// TIA Portal V20 export
FUNCTION_BLOCK "GM_ReceiveFData"   // FB116, LAD
TITLE = Template: GM sending data
// Template v0.1
// stored: MemoryReserve 100, Namespace Safety, SetENOAutomatically false
   VAR_INPUT
      Connection_ID_Send : Word;
      Connection_ID_Receive : Word;
      Send_Ack_Rcv_Length : UInt;
      Receive_Rcv_Length : UInt;
   END_VAR
   VAR_IN_OUT
      RcvBuffer : Array[0..1, 0..121] of Byte;   // Temporary receive buffer: Max Rcv-Array of F-Link Communication Length = 122 Bytes
      ReceivedData : Array[0..121] of Byte;   // Received raw data from PLC 2
      ReceivedAck : Array[0..121] of Byte;   // Received acknowledge data for communication PLC 1 to PLC 2
   END_VAR
   VAR
      instTRcvAck { S7_SetPoint := 'True'} : TRCV;   // Receive acknowledge data from PLC2
      instTRcvData { S7_SetPoint := 'True'} : TRCV;   // Receive data from PLC2
      statErrorRcvAck { S7_SetPoint := 'True'} : Word;   // variable for saving the status of TRCV block in case of error
      statErrorRcvData : Word;   // variable for saving the status of TRCV block in case of error
   END_VAR
BEGIN

REGION Network 1: Receive ACK_RCV_ARRAY from Plc1ToPlc2 Communication / Receive Acknowledge signal from partner
   // receive ack. signal from each station
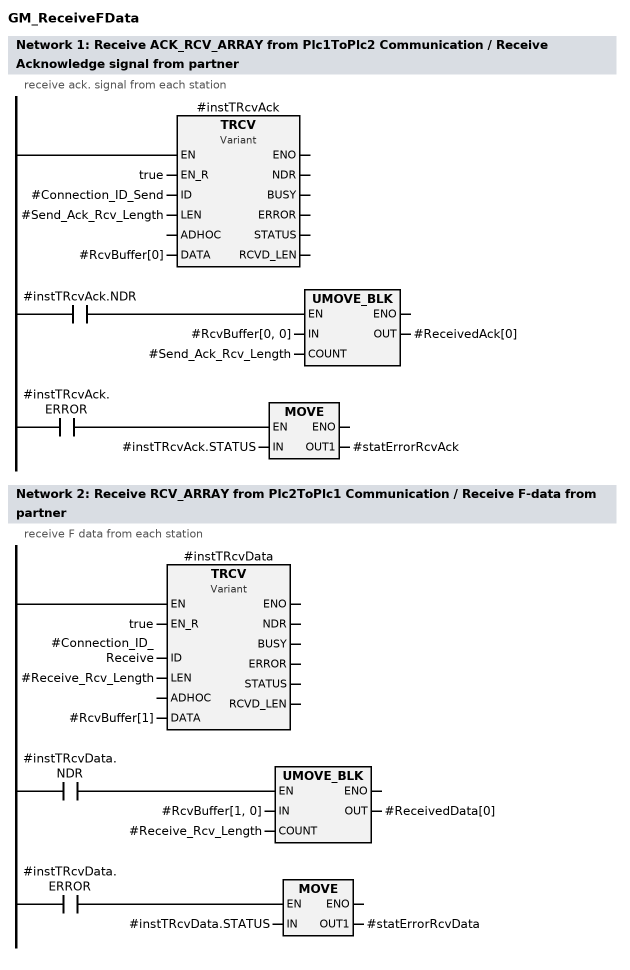
   #instTRcvAck(EN_R := true, ID := #Connection_ID_Send, LEN := #Send_Ack_Rcv_Length, DATA := #RcvBuffer[0]);   // TRCV
   IF #instTRcvAck.NDR THEN
       UMOVE_BLK(IN := #RcvBuffer[0, 0], COUNT := #Send_Ack_Rcv_Length, OUT => #ReceivedAck[0]);
   END_IF;
   IF #instTRcvAck.ERROR THEN #statErrorRcvAck := #instTRcvAck.STATUS; END_IF;
END_REGION

REGION Network 2: Receive RCV_ARRAY from Plc2ToPlc1 Communication / Receive F-data from partner
   // receive F data from each station
   #instTRcvData(EN_R := true, ID := #Connection_ID_Receive, LEN := #Receive_Rcv_Length, DATA := #RcvBuffer[1]);   // TRCV
   IF #instTRcvData.NDR THEN
       UMOVE_BLK(IN := #RcvBuffer[1, 0], COUNT := #Receive_Rcv_Length, OUT => #ReceivedData[0]);
   END_IF;
   IF #instTRcvData.ERROR THEN #statErrorRcvData := #instTRcvData.STATUS; END_IF;
END_REGION
END_FUNCTION_BLOCK
